FUNCTION_BLOCK FB_AUT_180 EXTENDS FB_AUT_ABSTRACT
(****************************************************************************)
(*	POU_AUT_zxx			Bausteinaufrufe Station	zxx							*)
(*	Status				ungetestet											*)
(*  Version:			1.0													*)
(*	Beschrieb:																*)
(*																			*)
(*	Abläufe:			FB_ABLzxxA		Hauptablauf							*)
(*																			*)
(*																			*)
(* 	25.09.2019/Dj															*)
(****************************************************************************)
(*	dd.mm.yyyy   KZ    x.y			Beschrieb								*)
(****************************************************************************)
VAR_INPUT
    (* spezifische Eingänge *)

END_VAR
VAR_OUTPUT
    (* spezifische Ausgänge *)

END_VAR
VAR
    (* Bausteine *)
    fb_Pnp    : FB_ABL_180_Pnp;

    fb_stat : FB_AUT_Statistics;

END_VAR

(*******************************************************************)
(* Timer *)
(*******************************************************************)

(*******************************************************************)
(* Flanken / Merker *)
(*******************************************************************)
//MANU CYCLE
IF (enIN_State = StateMANU) AND xIN_ManuCycle THEN
    xManuCycle := TRUE;
END_IF;

IF (enIN_State <> StateMANU) OR xOUT_Done THEN
    xManuCycle := FALSE;
END_IF

//NEXT STEP
xNextStep := (enIN_State > StateSTEP) OR
             ((enIN_State = StateSTEP) AND xIN_Step) OR
             ((enIN_State = StateMANU) AND xManuCycle);

//RESET
xReset := (enIN_State < StateREADY) AND (enIN_State <> StateINIT) AND NOT xManuCycle;

(*******************************************************************)
(* Bausteinaufrufe Abläufe *)
(*******************************************************************)

xRelease := MAIN.MoverMan.IsProcessUsed(THIS^);

fb_Pnp(xIN_Reset          := xReset,
       xIN_Init           := xIN_Init,
       xIN_Quit           := xIN_Quit,
       xIN_Start          := enIN_State >= enState.StateLEER AND xRelease,
       xIN_Sperre         := NOT xIN_On,
       xIN_NextStep       := xNextStep,
       xIN_AlarmAktiv     := xIN_AlarmAktiv,
       xIN_DryCycle       := xIN_DryCycle,
       xIN_RestartCYCL    := enIN_State >= enState.StateLEER,
       enIN_State         := enIN_State,
       tIN_Timeout        := tIN_Timeout,
       pxFG_Freigabe      := ADR(xRelease),
       Mover              := THIS^.Mover,
       xIN_PceReadyToPick := TRUE);

fb_stat(xIN_Enable  := enIN_State = enState.StateAUTO,
        xIN_Waiting := fb_Pnp.xOUT_Wait,
        xIN_Running := (fb_Pnp.iOUT_Step >= ST180_Pnp_e.START) AND
                       (fb_Pnp.iOUT_Step <= ST180_Pnp_e.DONE),
        // Since we use a mover system, a cycle is done when we are waiting on a mover
        xIN_Done := fb_Pnp.iOUT_Step = ST180_Pnp_e.waitOnMover);

(*******************************************************************)
(* Mover reset flags *)
(*******************************************************************)

(*******************************************************************)
(* OUTPUT *)
(*******************************************************************)
xOUT_InitDone := fb_Pnp.xOUT_InitDone;
xOUT_Ready    := fb_Pnp.xOUT_Ready;
xOUT_Done     := fb_Pnp.xOUT_Done;
xOUT_ErrFlag  := fb_Pnp.xOUT_ErrFlag;
xOUT_Wait     := fb_Pnp.xOUT_Wait;
xOUT_AlarmST  := xOUT_ErrFlag;

(*******************************************************************)
(* Bausteinaufruf Error Station *)
(*******************************************************************)
// POU_ERR_VORLAGE(xIN_QUIT:=xIN_Quit , pstrArIN_ALARM:=ADR(HMI.strArALARM[1]));

(* % of completion of the process *)
PROPERTY iCompletionPC : INT
GET
iCompletionPC := THIS^.fb_Pnp.iOUT_ProcessCompletion;
END_GET
END_PROPERTY

PROPERTY ProcessExecution : ProcessExecution_e
GET
ProcessExecution := THIS^._ProcessExecution;
END_GET
SET
THIS^._ProcessExecution := ProcessExecution;
END_SET
END_PROPERTY

PROPERTY xBusy : BOOL
GET
xBusy := THIS^.fb_Pnp.xOUT_Busy;
END_GET
SET
END_SET
END_PROPERTY

PROPERTY xDone : BOOL
GET
xDone := THIS^.fb_Pnp.xOUT_Ready OR THIS^.fb_Pnp.xOUT_Done;
END_GET
END_PROPERTY

PROPERTY xMoverPathFree : BOOL
GET
xMoverPathFree := THIS^.fb_Pnp.xOUT_MoverFree OR THIS^.fb_Pnp.xOUT_Ready OR THIS^.fb_Pnp.xOUT_Done;
END_GET
END_PROPERTY

PROPERTY xMoverShouldLeave : BOOL
GET
xMoverShouldLeave := THIS^.fb_Pnp.iOUT_Step = ST180_Pnp_e.SYNC_MOVER_LEAVE;
END_GET
END_PROPERTY

END_FUNCTION_BLOCK

(* stored: Version 1.1.0.1, ProductVersion 3.1.4024.6
   POU FB_AUT_180: Id {1e8b7016-d446-49ee-9e1a-ab246c4a32ea}, SpecialFunc None
   Property iCompletionPC: Id {e025fa00-2775-4351-99de-bf79b8c7a85b}
   Get Get: Id {5e103c89-c1bc-4ba6-b7f3-865974813690}
   Property ProcessExecution: Id {c643cedd-d4fb-452b-9b65-8b4cee8eb6aa}
   Get Get: Id {38c41f7c-42ac-43c3-b452-229bd8076f09}
   Set Set: Id {e304c586-3987-47ea-8d1a-0a2b91f58643}
   Property xBusy: Id {f8fde9ef-cb14-4859-a13a-42042673975d}
   Get Get: Id {dc445834-586a-46b9-b051-40101e6c7778}
   Set Set: Id {53e2ccfb-4bc1-4406-a559-67e7047db0bd}
   Property xDone: Id {b6783e61-268a-4b4b-80c9-2005d16ff7e3}
   Get Get: Id {dec483ca-5552-470c-9f82-790993b6553b}
   Property xMoverPathFree: Id {c367e1e3-f584-42a4-a5e0-d7145c0bbd40}
   Get Get: Id {16ab4e4f-5778-4736-8111-53d76adec3f9}
   Property xMoverShouldLeave: Id {c2765c2b-0342-46a3-9536-d7b8a8df48e2}
   Get Get: Id {3916cd15-ec58-4a7f-aef3-24f4bfa3a96e} *)
